TYPE ST_LSS :
STRUCT
	
	State						: E_LSS_State;
	CMD							: ST_GeneralStationCMD;	
	Status						: ST_StationStatus;
	
END_STRUCT
END_TYPE

(* stored: Version 1.1.0.1, ProductVersion 3.1.4026.18
   DUT ST_LSS: Id {6fd7b079-1432-4b2f-b82c-e9b72471f28e} *)
